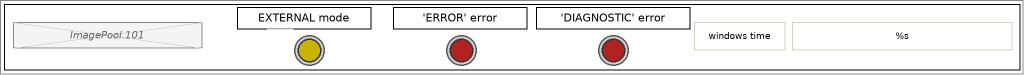
VISUALIZATION MenuTop  // 1024x75
    RoundedRectangle (4,4 1016x66)
    Lamp1 (292,33 35x35), variable: MAIN.fbKRC_AutomaticExternal.IO_ACTCONF, style: Lamp-Lamp1-Yellow
    Lamp1 (444,33 35x35), variable: MAIN.fbKRC_Error.Error, style: Lamp-Lamp1-Red
    Textfield (792,22 220x28), "%s", text variable: GVL_PLC.String_WindowsTime
    Textfield (694,22 91x28), "windows time"
    Lamp1 (596,33 35x35), variable: MAIN.fbKRC_Diag.Error, style: Lamp-Lamp1-Red
    RoundedRectangle (237,7 134x22), "EXTERNAL mode"
    RoundedRectangle (393,7 134x22), "'ERROR' error"
    RoundedRectangle (536,7 154x22), "'DIAGNOSTIC' error"
    Image (13,22 189x26), image: ImagePool.101
    Image (267,28 26x1)
END_VISUALIZATION

(* stored: Version 1.1.0.1, ProductVersion 3.1.4024.10
   Visu MenuTop: Id {8f5b1f6a-8efc-4a8d-a84b-d10046e43a4e} *)
